(* PLC project Unnamed, Unknown Unnamed 1 *)
(* stored: creationDateTime 2025-06-21T16:09:36, modificationDateTime 2025-06-21T16:36:18 *)

PROGRAM sel_pou
  VAR
    input1 AT %IX100.0 : BOOL;
    input2 AT %IX100.1 : BOOL;
    reset AT %IX100.2 : BOOL;
    load AT %IX100.3 : BOOL;
    output1 AT %QX100.0 : BOOL;
    output2 AT %QX100.1 : BOOL;
  END_VAR
  VAR
    R_TRIG0 : R_TRIG;
    CTU0 : CTU;
    R_TRIG1 : R_TRIG;
    CTU1 : CTU;
  END_VAR
  VAR  (* added by the conversion: wires and edge detectors of the diagram *)
    R_TRIG1_2 : R_TRIG;
    R_TRIG2 : R_TRIG;
  END_VAR

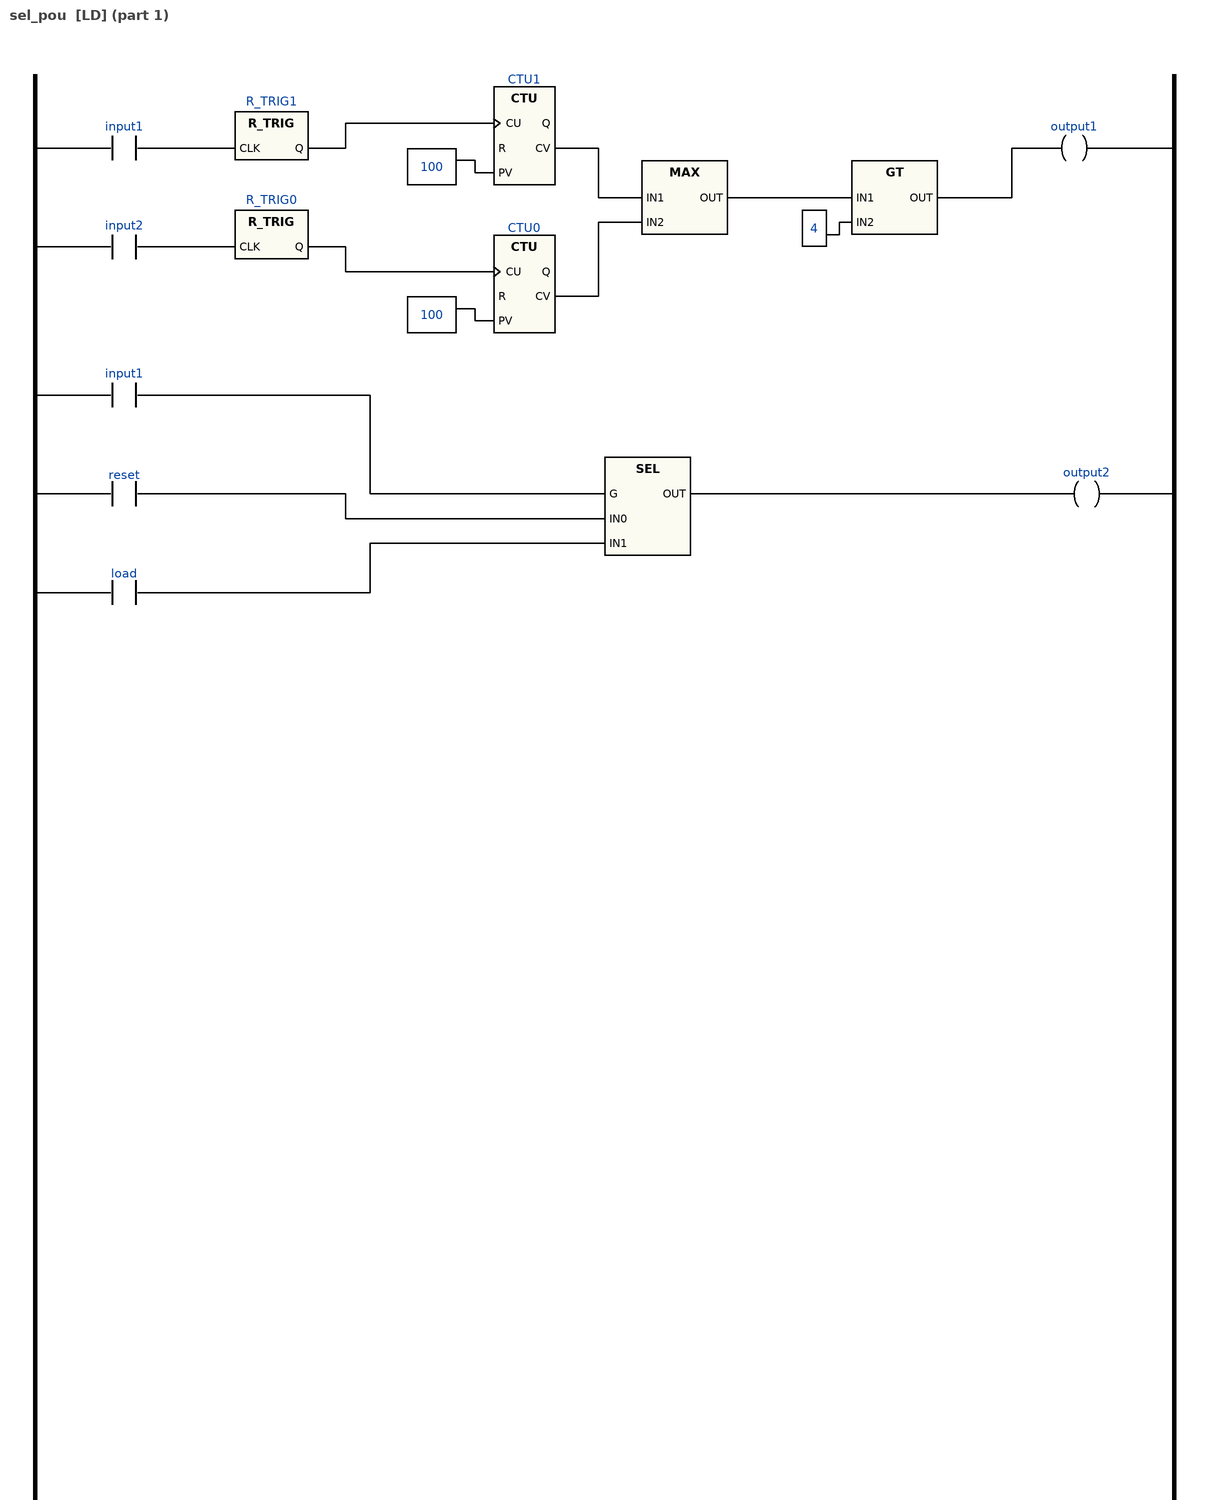
(* LD diagram, written out as Structured Text *)
R_TRIG1(CLK := input1);
R_TRIG1_2(CLK := R_TRIG1.Q);
CTU1(CU := R_TRIG1_2.Q, PV := 100);
R_TRIG0(CLK := input2);
R_TRIG2(CLK := R_TRIG0.Q);
CTU0(CU := R_TRIG2.Q, PV := 100);
output1 := MAX(CTU1.CV, CTU0.CV) > 4;
output2 := SEL(input1, reset, load);
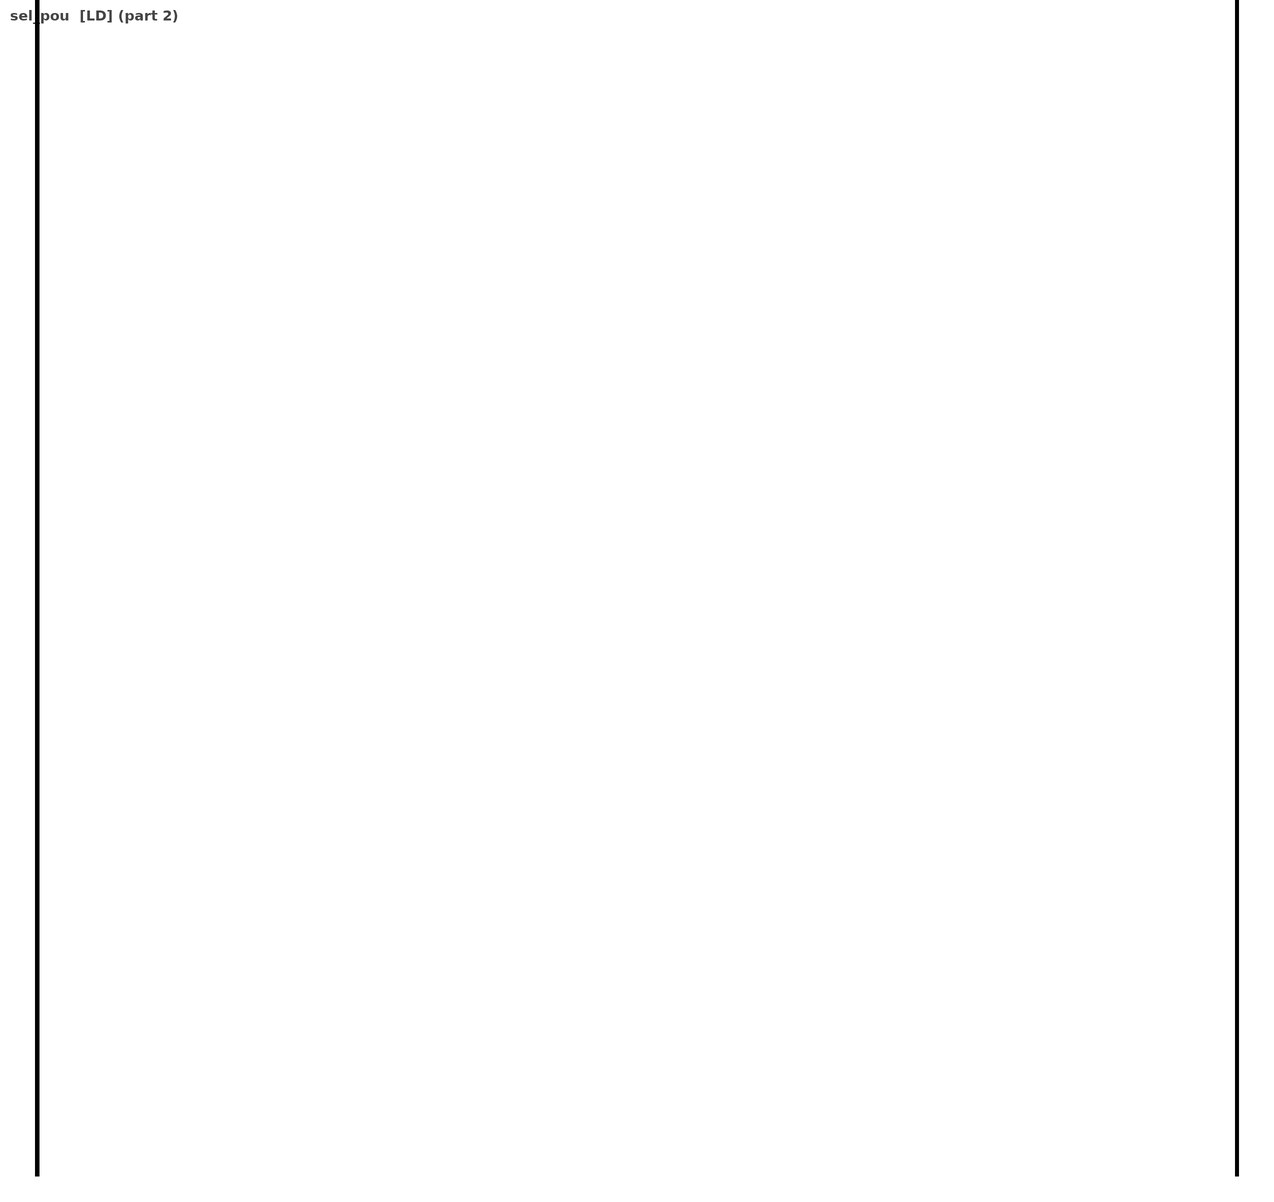
END_PROGRAM

CONFIGURATION Config0
  RESOURCE Res0 ON PLC
    TASK task0(INTERVAL := T#20ms, PRIORITY := 0);
    PROGRAM instance0 WITH task0 : sel_pou;
  END_RESOURCE
END_CONFIGURATION
